// TIA Portal V19 export
TYPE "FeedMachine_COut"
// stored: Access Published
   STRUCT
      Infeed_ReqON : Bool;
      CtrlSafe : Bool;
      Standstill : Bool;
      Bwd_CheckNext : Bool;
      Fwd_CheckNext : Bool;
      Bwd_VelZero : Bool;
      Bwd_Running : Bool;
      Fwd_VelZero : Bool;
      Fwd_Running : Bool;
      ActualVelocity : LReal;   // [mm/min]
      TargetVelocity : LReal;
      MaxVelocity : LReal;
   END_STRUCT;
END_TYPE
